(* IEC 61131-3 sources: LStream-JSON-XML/src/LStream/Utilities, 3 files *)

(* ---- LStream_FindStringInByteCharArrayAdv.st ---- *)
//REGION BLOCK INFO HEADER
//===============================================================================
  // SIEMENS AG / (c)Copyright 2021
  //-------------------------------------------------------------------------------
  // Title:            LStream_FindStringInByteCharArrayAdv
  // Comment/Function: Searches for a specified string within an array of char
  // Library/Family:   LStream
  // Author:           DI FA S SUP E&C
  // Tested with:      S7-1500 V2.8
  // Engineering:      TIA Portal V16
  // Restrictions:     --
  // Requirements:     --
  //-------------------------------------------------------------------------------
  // Change log table:
  // Version  | Date       | Expert in charge | Changes applied
  //----------|------------|------------------|------------------------------------
  // 01.00.00 | 2021-03-10 |DI FA S SUP E&C   | First released version
  //===============================================================================

//END_REGION

USING System.Strings;
USING System.Math;
NAMESPACE Simatic.Ax.LStream.Utilities
  FUNCTION LStream_FindStringInByteCharArrayAdv : DINT  //Returns the index of found string
    VAR_INPUT
      /// Text that is searched for
      searchFor : STRING;
      /// Start position in array   //CHANGE TO UDINT;
      startPosition : DINT;
    END_VAR
    VAR_IN_OUT
      /// Array of Char to search in
      searchIn : ARRAY[*] of BYTE;
    END_VAR
    VAR_TEMP
      /// Lower bound of given array
      tempLowerBound : DINT;
      /// Number of elements in given array
      tempNumElements : UDINT;
      /// Length of text that is searched for
      tempLenSearchFor : INT;
      /// Position in array during search (0-based)
      tempPosInArray : DINT;
      /// Position in working string during search
      tempPosInString : INT;
      /// Temporary string to work with
      tempString : STRING;
    END_VAR
    VAR CONSTANT
      /// Constant for first array dimension
      FIRST_DIM : USINT := USINT#1;
      /// Max.length of String
      MAX_LEN_STRING : UINT := UINT#254;
    END_VAR

    // Initialization
    tempPosInString := 0;
    tempPosInArray := startPosition;
    tempLenSearchFor := LengthOf(value := searchFor);
    LStream_FindStringInByteCharArrayAdv := -1;

    // Get number of elements

    tempLowerBound := LOWER_BOUND(searchIn, FIRST_DIM);
    tempNumElements := TO_UDINT(UPPER_BOUND(searchIn,FIRST_DIM) - tempLowerBound + 1);

    IF (TO_LINT(tempPosInArray) > tempNumElements) THEN      //Convert to LINT to ensure that if i convert to UINT is not out of range
      RETURN;
    END_IF;

    // Search for beginning of text until something was found and
    // as long as the index is less than the array size / number of elements in array
    WHILE ((tempPosInString <= 0) AND (TO_UDINT(tempPosInArray) < tempNumElements)) DO
      // Convert Chars to String
      CharsToString(chars := searchIn,
                    startPosition := tempPosInArray,
                    length:= TO_UINT(Min(MAX_LEN_STRING, tempNumElements)),
                    result => tempString);

      // Search for text at beginning
      tempPosInString := PositionOf(value := tempString, seekValue := searchFor);      //CHECK HOW TO IMPLEMENT

      // Keyword was found
      IF tempPosInString > 0 THEN
        // Output position of string
        LStream_findStringInByteCharArrayAdv := tempLowerBound + tempPosInArray + tempPosInString -1;
        EXIT;
      ELSE
        // Otherwise continue search in next string minus length of text at beginning to ensure
        // keywords are not broken up at the end of a string and thus missed
        tempPosInArray := tempPosInArray + TO_INT(MAX_LEN_STRING) - tempLenSearchFor;
      END_IF;
    END_WHILE;

  END_FUNCTION
END_NAMESPACE

(* ---- LStream_WriteOutString.st ---- *)
USING System.Strings;
USING System.Serialization;
NAMESPACE Simatic.Ax.LStream.Utilities
    FUNCTION LStream_WriteOutString : INT  //Offset after the data has been written; -1 if there would have been an overflow
        VAR_INPUT
            /// Position in the array to start writing
            offset : UINT;
        END_VAR
        VAR_IN_OUT
            /// The string that has to be written to the byte array
            toWrite : STRING;
            /// The byte representation of the XML to write into
            xmlByteArray : ARRAY[*] of BYTE;
        END_VAR
        VAR_TEMP
            /// The upper bound index of the XML Array
            tempXmlUpperBound : DINT;
            /// Amount of characters written to the char array
            tempCountWritten : UDINT;
            tempOffsetArray : ARRAY[0..255] of BYTE;
            Index : INT;
        END_VAR
        VAR CONSTANT
            /// Return value, if the write would be out of bounds, no write happens
            RETURN_OUT_OF_BOUNDS : INT := -1;
            /// Max.length of String
            MAX_LEN_STRING : UINT := UINT#254;
        END_VAR

        tempXmlUpperBound := UPPER_BOUND(xmlByteArray, 1);

        LStream_WriteOutString := RETURN_OUT_OF_BOUNDS;

        IF ((TO_UINT(LengthOf(toWrite)) + offset) > tempXmlUpperBound) THEN
            RETURN;
        END_IF;

        //add information to xml byte array

        // //SERIALIZE
        // tempCountWritten := Serialize(offset := offset, value := toWrite, buffer :=  xmlByteArray); //error due to serialize writing size in output byte array

        // //fixed serialize
        tempCountWritten := Serialize(offset := UDINT#0, value := toWrite, buffer := tempOffsetArray); //NOT WORKING BECAUSE STRING SIZE IS WRITTEN IN FIRST POSITION OF OUTPUT ARRAY
        //WRITE INTO OUTPUT ARRAY WITH AN OFFSET TO AVOID WRITING STRING SIZE - USE SIZE IN FIRST BYTE FOR LIMIT NUMBER OF ITERATIONS
        FOR Index := 0 TO TO_INT(tempOffsetArray[0]) - 1 DO
            xmlByteArray[TO_INT(offset) + Index] := tempOffsetArray[Index + 1];
        END_FOR;

        /*Strg_TO_Chars(Strg := toWrite,
                    pChars := offset,
                    Cnt => tempCountWritten,
                    Chars := xmlByteArray);
        */
        //move index of byte array
        LStream_WriteOutString := LStream_WriteOutString + TO_INT(tempCountWritten) - 1;

    END_FUNCTION
  END_NAMESPACE

(* ---- StringToByteArray.st ---- *)
USING System.Strings;
NAMESPACE Simatic.Ax.LStream.Utilities
    FUNCTION StringToByteArray : BOOL
        VAR_INPUT
            string1 : STRING;
            /// Optional
            string2 : STRING := '';
            /// Optional
            string3 : STRING := '';
            /// Optional
            string4 : STRING := '';
        END_VAR

        VAR_IN_OUT
            /// Ensure this array is large enough to hold all bytes
            byteArray : ARRAY[0..10000] OF BYTE;
        END_VAR

        VAR
            totalLength : INT := 0;
            stringLength : INT;
            byteIndex : INT := 0;
            SizeOfByteArray : DINT := 10000;
            i : INT;
        END_VAR

        // Process string1
        IF string1 <> '' THEN
            stringLength := LengthOf(string1);
            IF (totalLength + stringLength) > SizeOfByteArray THEN
                StringToByteArray := FALSE; // Not enough space in the byte array
                RETURN;
            END_IF;

            FOR i := 1 TO stringLength DO
                byteArray[byteIndex] := TO_BYTE(TO_USINT(string1[i]));
                byteIndex := byteIndex + 1;
            END_FOR;
            totalLength := totalLength + stringLength;
        END_IF;

        // Process string2
        IF string2 <> '' THEN
            stringLength := LengthOf(string2);
            IF (totalLength + stringLength) > SizeOfByteArray THEN
                StringToByteArray := FALSE; // Not enough space in the byte array
                RETURN;
            END_IF;

            FOR i := 1 TO stringLength DO
                byteArray[byteIndex] := TO_BYTE(TO_USINT(string2[i]));
                byteIndex := byteIndex + 1;
            END_FOR;
            totalLength := totalLength + stringLength;
        END_IF;

        // Process string3
        IF string3 <> '' THEN
            stringLength := LengthOf(string3);
            IF (totalLength + stringLength) > SizeOfByteArray THEN
                StringToByteArray := FALSE; // Not enough space in the byte array
                RETURN;
            END_IF;

            FOR i := 1 TO stringLength DO
                byteArray[byteIndex] := TO_BYTE(TO_USINT(string3[i]));
                byteIndex := byteIndex + 1;
            END_FOR;
            totalLength := totalLength + stringLength;
        END_IF;

        // Process string4
        IF string4 <> '' THEN
            stringLength := LengthOf(string4);
            IF (totalLength + stringLength) > SizeOfByteArray THEN
                StringToByteArray := FALSE; // Not enough space in the byte array
                RETURN;
            END_IF;

            FOR i := 1 TO stringLength DO
                byteArray[byteIndex] := TO_BYTE(TO_USINT(string4[i]));
                byteIndex := byteIndex + 1;
            END_FOR;
            totalLength := totalLength + stringLength;
        END_IF;

        // If all strings were successfully processed
        StringToByteArray := TRUE;
        RETURN;
    END_FUNCTION

END_NAMESPACE
